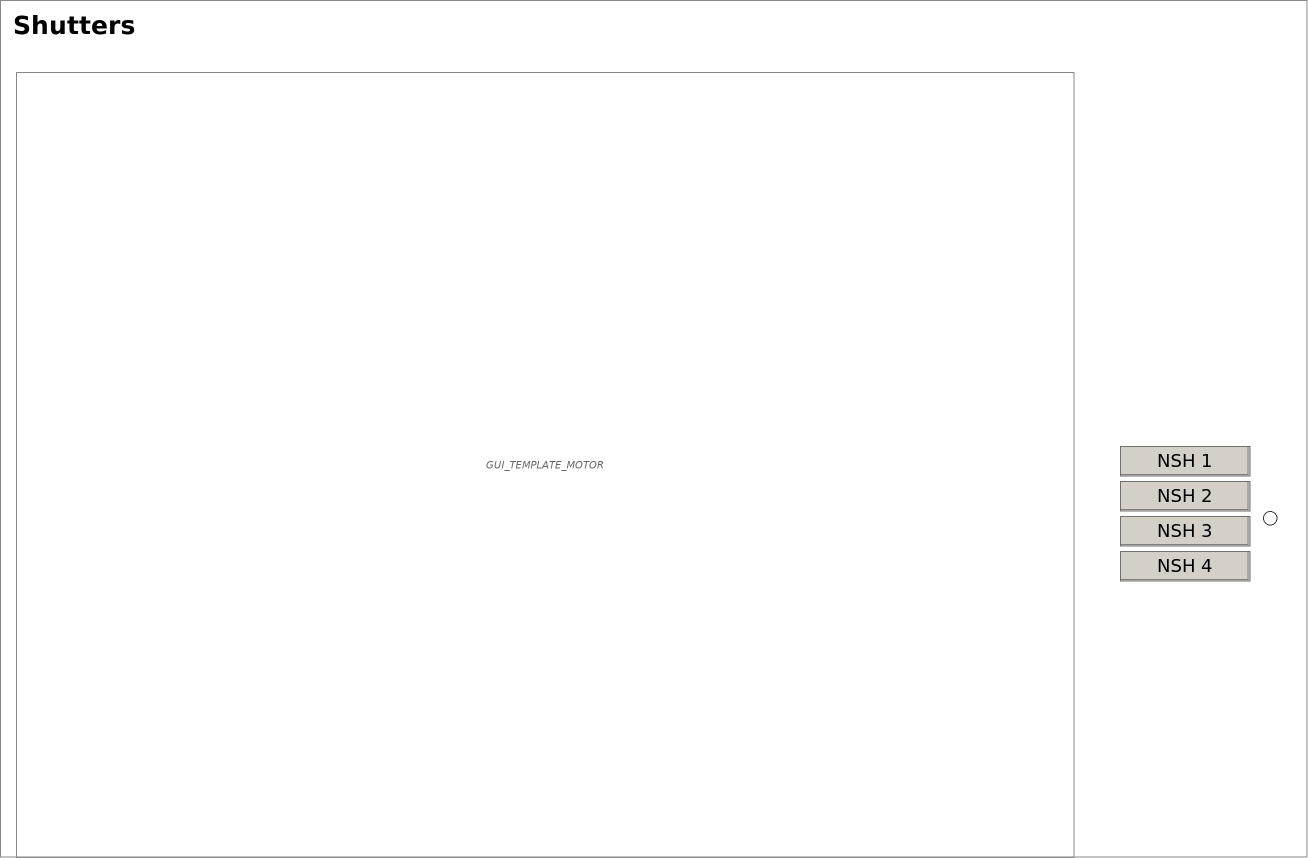
VISUALIZATION VISU_HMI_SHUTTERS  // 1308x858
    Label (10,10 199x30), "Shutters"
    RadioButton (1261,448 47x140), variable: MAIN.nott_ics.Shutters.guiShutterIndex-1
        Areas[0]: Text=Radiobutton
        Areas[1]: Text=Radiobutton
    Button (1120,446 130x30), "NSH 1"
        OnMouseClick: execute { MAIN.nott_ics.Shutters.guiShutterIndex := 1; }
    Button (1120,481 130x30), "NSH 2"
        OnMouseClick: execute { MAIN.nott_ics.Shutters.guiShutterIndex := 2; }
    Button (1120,516 130x30), "NSH 3"
        OnMouseClick: execute { MAIN.nott_ics.Shutters.guiShutterIndex := 3; }
    Button (1120,551 130x30), "NSH 4"
        OnMouseClick: execute { MAIN.nott_ics.Shutters.guiShutterIndex := 4; }
    Frame (16,72 1058x786)
        shows GUI_TEMPLATE_MOTOR(m_Instance := MAIN.nott_ics.Shutters.ptrShutters[MAIN.nott_ics.Shutters.guiShutterIndex]^)
END_VISUALIZATION

(* stored: Version 1.1.0.1, ProductVersion 3.1.4024.15
   Visu VISU_HMI_SHUTTERS: Id {bc7ead1a-79ad-498a-88b1-c825494753c4} *)
